// TIA Portal V20 export
// export: Created 2025-09-12T17:57:00.0000000Z, ExportSetting WithDefaults
TYPE "UDT200_EM_Cooling"
   STRUCT
      HP_Switch_DI : Bool;   // Digital Input: High-pressure refrigerant switch (`True` = Fault).
      LP_Switch_DI : Bool;   // Digital Input: Low-pressure refrigerant switch (`True` = Fault).
      Freeze_Stat_DI : Bool;   // Digital Input: Freeze-stat on coil (`True` = Fault).
      Compressor_Cmd_DO : Bool;   // Digital Output: Command to start/stop the compressor.
      Min_Run_Time_Sec : Time;   // Minimum compressor run time to prevent short-cycling (e.g., `T#3m`).
      Min_Off_Time_Sec : Time;   // Minimum compressor off time to prevent short-cycling (e.g., `T#3m`).
      HP_Fault_Alm : Bool;   // Alarm: High-pressure fault.
      LP_Fault_Alm : Bool;   // Alarm: Low-pressure fault.
      Freeze_Stat_Alm : Bool;   // Alarm: Freeze-stat tripped.
   END_STRUCT;
END_TYPE
